// TIA Portal V20 export
// export: Created 2026-07-10T11:12:23.3722674Z, ExportSetting WithDefaults, DisplayName Totally Integrated Automation Portal, DisplayVersion V20, DisplayName TIA Portal Openness, DisplayVersion V20, DisplayName TIA Portal Version Control Interface, DisplayVersion V20, DisplayName STEP 7 Professional, DisplayVersion V20, DisplayName STEP 7 Safety, DisplayVersion V20, DisplayName WinCC Basic/Comfort/Advanced, DisplayVersion V20, DisplayName WinCC Unified, DisplayVersion V20
FUNCTION_BLOCK "Inputs"   // FB4, SCL
{ S7_Optimized_Access := 'TRUE' }
VERSION : 0.1
// stored: AutoNumber true, IsIECCheckEnabled false, IsRetainMemResEnabled false, MemoryReserve 100, SetENOAutomatically false, UDAEnableTagReadback false
   VAR
      AIHandlers { S7_SetPoint := 'True'} : Array[0..5] of "AIHandler";
      WeightHandlers { S7_SetPoint := 'True'} : Array[0..1] of "WeightHandler";
      ErrorRCV1 { S7_SetPoint := 'True'} : Bool;
      ErrorRCV2 { S7_SetPoint := 'True'} : Bool;
   END_VAR
BEGIN
   #AIHandlers[0](
                  Value := "AI0AV",
                  ValueMin := 0,
                  ValueMax := 27648,
                  ValueOffset := "MB".Table.AIOffsetCH0,
                  OutputMin := "MB".Table.AIValueMinCH0,
                  OutputMax := "MB".Table.AIValueMaxCH0,
                  TimeBase := "MB".Table.AITimeBaseCH0,
                  Output => "MB".Table.WaterInPressureValue);
   #AIHandlers[1](
                  Value := "AI1AV",
                  ValueMin := 0,
                  ValueMax := 27648,
                  ValueOffset := "MB".Table.AIOffsetCH1,
                  OutputMin := "MB".Table.AIValueMinCH1,
                  OutputMax := "MB".Table.AIValueMaxCH1,
                  TimeBase := "MB".Table.AITimeBaseCH1,
                  Output => "MB".Table.RCV1LevelValue);
   #AIHandlers[2](
                  Value := "AI2AV",
                  ValueMin := 0,
                  ValueMax := 27648,
                  ValueOffset := "MB".Table.AIOffsetCH2,
                  OutputMin := "MB".Table.AIValueMinCH2,
                  OutputMax := "MB".Table.AIValueMaxCH2,
                  TimeBase := "MB".Table.AITimeBaseCH2,
                  Output => "MB".Table.RCV2LevelValue);
   #AIHandlers[3](
                  Value := "AI3AV",
                  ValueMin := 0,
                  ValueMax := 27648,
                  ValueOffset := "MB".Table.AIOffsetCH3,
                  OutputMin := "MB".Table.AIValueMinCH3,
                  OutputMax := "MB".Table.AIValueMaxCH3,
                  TimeBase := "MB".Table.AITimeBaseCH3,
                  Output => "MB".Table.WaterOutPressureValue);
   // #AIHandlers[4](
   //                Value := "AI4AV",
   //                ValueMin := 5320,
   //                ValueMax := 27648,
   //                ValueOffset := "MB".Table.AIOffsetCH4,
   //                OutputMin := "MB".Table.AIValueMinCH4,
   //                OutputMax := "MB".Table.AIValueMaxCH4,
   //                TimeBase := "MB".Table.AITimeBaseCH4,
   //                Output => );

   #ErrorRCV1 := #AIHandlers[1].Error;
   #ErrorRCV2 := #AIHandlers[2].Error;


   CASE "MB".Table.DampersSyncMode OF
       1:
           "MB".Table.RCV1LevelValue := "MB".Table.RCV1LevelValue;
           "MB".Table.RCV2LevelValue := "MB".Table.RCV1LevelValue;
           #ErrorRCV2 := #ErrorRCV1;
       2:
           "MB".Table.RCV1LevelValue := "MB".Table.RCV2LevelValue;
           "MB".Table.RCV2LevelValue := "MB".Table.RCV2LevelValue;
           #ErrorRCV1 := #ErrorRCV2;
   END_CASE;
END_FUNCTION_BLOCK
